{attribute 'qualified_only'}
{attribute 'to_string'}
TYPE E_OuterLoopSM_States :
(
	Setup := 0,
	Operational,
	DisablingInactive,
	DisablingError,
	Inactive,
	DisabledError,
	UserDisabled,
	DisablingUserDisable
) UINT := Setup
;
END_TYPE

(* stored: Version 1.1.0.1, ProductVersion 3.1.4024.12
   EnumerationTextList E_OuterLoopSM_States: Id {08f83fa9-d361-490f-bd27-af917550d7d1} *)
